{attribute 'qualified_only'}
VAR_GLOBAL
	fbCylinder	: FB_Cylinder(refExtendOut := GVL_Io.bExtendOut, refRetractOut := GVL_Io.bRetractOut);
	fbStation	: FB_Station;
	fbDerived	: FB_StationDerived;
END_VAR

(* stored: Version 1.1.0.1, ProductVersion 3.1.4024.12
   GVL GVL_System: Id {db2ff4ce-1d8a-4d04-8167-a635fc81f165} *)
